KUKA KRL program: letter_t_surname.src

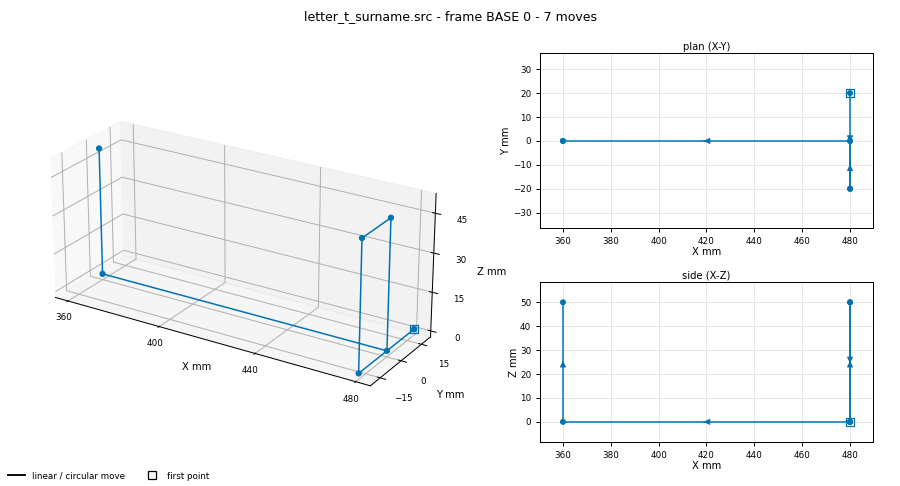
[picture p0: tool path of letter_t_surname.src in frame BASE 0, 7 of 10 moves have a stored position in this frame; points joined in program order, loops and branches not executed]
&ACCESS RVP
&REL 1
&PARAM TEMPLATE = C:\KRC\Roboter\Template\vorgabe
&PARAM EDITMASK = *
DEF letter_t_surname ( )

;FOLD Initialise and set default speed
BAS (#INITMOV,0)
BAS (#VEL_PTP,100)
BAS (#ACC_PTP,20)
$VEL.CP=0.2
BAS (#TOOL,0)
BAS (#BASE,0)
;ENDFOLD

$ADVANCE = 5

; Program generated by RoboDK v5.2.5 for KUKA KR 4 R600 on 07/01/2025 12:35:32
; Using nominal kinematics.
$VEL.CP = 0.10000
PTP {A1 0.00000,A2 -101.70200,A3 131.55600,A4 0.00000,A5 60.14530,A6 0.00000,E1 0.00000}
PTP {A1 -2.86241,A2 -42.39960,A3 99.23040,A4 0.00000,A5 33.16920,A6 -2.86241,E1 0.00000}
$VEL.CP = 0.05000
LIN {X 480.000,Y 20.000,Z 0.000,A 0.000,B 0.000,C 0.000,E1 0.00000}
$VEL.CP = 0.07500
LIN {X 480.000,Y -20.000,Z 0.000,A 0.000,B 0.000,C 0.000,E1 0.00000}
$VEL.CP = 0.05000
LIN {X 480.000,Y -20.000,Z 50.000,A 0.000,B 0.000,C 0.000,E1 0.00000}
LIN {X 480.000,Y 0.000,Z 50.000,A 0.000,B 0.000,C 0.000,E1 0.00000}
LIN {X 480.000,Y 0.000,Z 0.000,A 0.000,B 0.000,C 0.000,E1 0.00000}
$VEL.CP = 0.07500
LIN {X 360.000,Y 0.000,Z 0.000,A 0.000,B 0.000,C 0.000,E1 0.00000}
$VEL.CP = 0.05000
LIN {X 360.000,Y 0.000,Z 50.000,A 0.000,B 0.000,C 0.000,E1 0.00000}
$VEL.CP = 0.10000
PTP {A1 0.00000,A2 -101.70200,A3 131.55600,A4 0.00000,A5 60.14530,A6 0.00000,E1 0.00000}
END
